(* IEC 61131-3 sources: plc_on_fpga_riscv_hybrid/RV_FPGA_PLC_IDE_Projects/PWM_TEST_var, 1 file *)

(* ---- PWM_TEST_var.il ---- *)
VAR
    Frequency   : INT
    Duty_Cycle   : INT
    PWM_1   : PWM
END_VAR

PROGRAM PWM_TEST_var
    Initialize_Variables :
        LD     2
        ST     Frequency
        LD     10
        ST     Duty_Cycle
    PWM_Function_Block :
        CAL PWM_1(
            F  := Frequency,
            DC := Duty_Cycle,
            Q  => %LEDG.0)
END_PROGRAM
